TYPE typeMotionScreenBtn :
STRUCT
		//define motion rows for HMI
	gMotionRow1btn: dutMotionRowButtons;
	gMotionRow2btn: dutMotionRowButtons;
	gMotionRow3btn: dutMotionRowButtons;
	gMotionRow4btn: dutMotionRowButtons;
	gMotionRow5btn: dutMotionRowButtons;
	gMotionRow6btn: dutMotionRowButtons;

	
END_STRUCT
END_TYPE

(* stored: Version 1.1.0.1, ProductVersion 3.1.4024.12
   DUT typeMotionScreenBtn: Id {0edfa3c2-52d5-4422-9e0c-babfdc41f9cf} *)
